PROGRAM MAIN
VAR
	_sampleComponentTests : SampleComponentTests;
END_VAR

END_PROGRAM

(* stored: Version 1.1.0.1, ProductVersion 3.1.4024.6
   POU MAIN: Id {773bf874-b264-48a0-a352-092af4113065}, SpecialFunc None *)
